FUNCTION_BLOCK L0_8070Service (* FAGOR 8070 CNC service FB *)
  (* Standard: 61499-2; Description: This FB is the entry point of the CNC service *)
  (* Version 0.0, 2014-09-01, EQUEROL, UJI *)
  (* Version 1.0, 2015-03-03, EQUEROL, UJI, Service rework *)
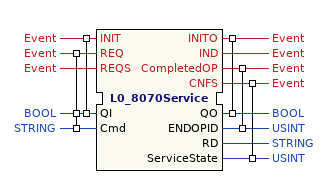
  EVENT_INPUT
    INIT WITH QI; (* Initialization Request *)
    REQ WITH QI, Cmd; (* Normal Execution Request *)
    REQS; (* Request Service state *)
  END_EVENT
  EVENT_OUTPUT
    INITO WITH QO; (* Initialization Confirm *)
    IND; (* Operation reception confirmation *)
    CompletedOP WITH ENDOPID; (* Completed operation event *)
    CNFS WITH ServiceState; (* Service State Confirmation *)
  END_EVENT
  VAR_INPUT
    QI : BOOL; (* Input event qualifier *)
    Cmd : STRING; (* String containing the actions to be executed *)
  END_VAR
  VAR_OUTPUT
    QO : BOOL; (* Output event qualifier *)
    ENDOPID : USINT; (* Operation end code *)
    RD : STRING; (* Service feedback data *)
    ServiceState : USINT; (* CNC Service state *)
  END_VAR
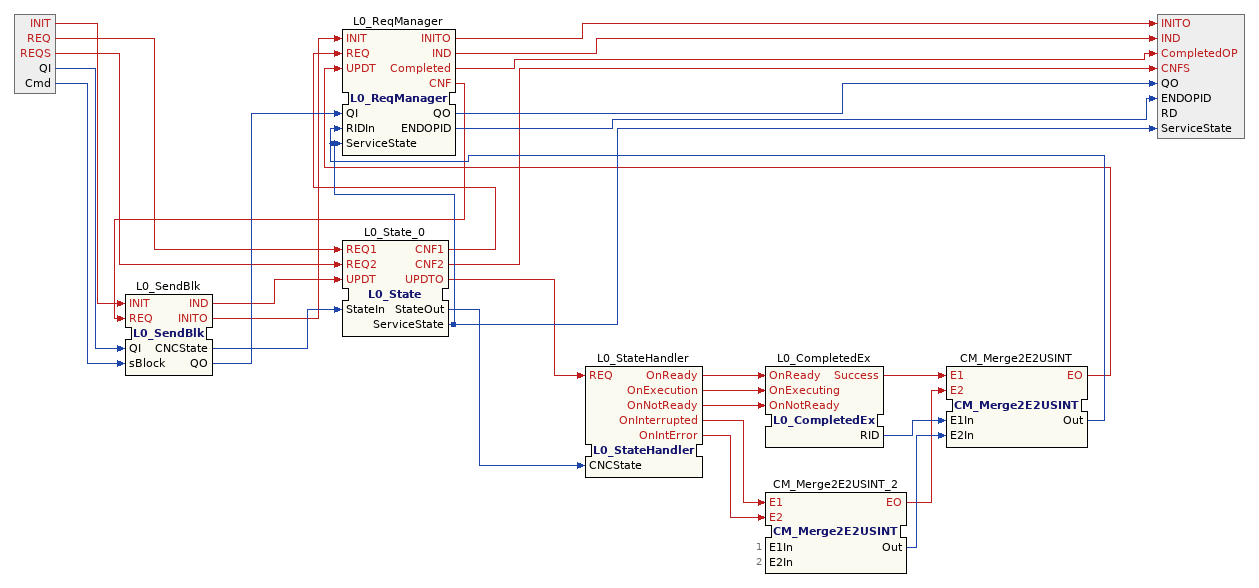
  FBS
    L0_SendBlk : L0_SendBlk;
    L0_StateHandler : L0_StateHandler;
    L0_CompletedEx : L0_CompletedEx;
    CM_Merge2E2USINT : CM_Merge2E2USINT;
    CM_Merge2E2USINT_2 : CM_Merge2E2USINT(E1In := 1, E2In := 2);
    L0_State_0 : L0_State;
    L0_ReqManager : L0_ReqManager;
  END_FBS
  EVENT_CONNECTIONS
    L0_StateHandler.OnReady TO L0_CompletedEx.OnReady;
    L0_StateHandler.OnExecution TO L0_CompletedEx.OnExecuting;
    L0_StateHandler.OnNotReady TO L0_CompletedEx.OnNotReady;
    L0_CompletedEx.Success TO CM_Merge2E2USINT.E1;
    CM_Merge2E2USINT_2.EO TO CM_Merge2E2USINT.E2;
    L0_StateHandler.OnInterrupted TO CM_Merge2E2USINT_2.E1;
    L0_StateHandler.OnIntError TO CM_Merge2E2USINT_2.E2;
    REQS TO L0_State_0.REQ2;
    L0_State_0.CNF2 TO CNFS;
    L0_State_0.UPDTO TO L0_StateHandler.REQ;
    L0_SendBlk.IND TO L0_State_0.UPDT;
    INIT TO L0_SendBlk.INIT;
    REQ TO L0_State_0.REQ1;
    L0_SendBlk.INITO TO L0_ReqManager.INIT;
    L0_State_0.CNF1 TO L0_ReqManager.REQ;
    CM_Merge2E2USINT.EO TO L0_ReqManager.UPDT;
    L0_ReqManager.INITO TO INITO;
    L0_ReqManager.CNF TO L0_SendBlk.REQ;
    L0_ReqManager.IND TO IND;
    L0_ReqManager.Completed TO CompletedOP;
  END_CONNECTIONS
  DATA_CONNECTIONS
    L0_CompletedEx.RID TO CM_Merge2E2USINT.E1In;
    CM_Merge2E2USINT_2.Out TO CM_Merge2E2USINT.E2In;
    L0_State_0.ServiceState TO ServiceState;
    L0_State_0.StateOut TO L0_StateHandler.CNCState;
    L0_SendBlk.CNCState TO L0_State_0.StateIn;
    QI TO L0_SendBlk.QI;
    L0_SendBlk.QO TO L0_ReqManager.QI;
    CM_Merge2E2USINT.Out TO L0_ReqManager.RIDIn;
    L0_ReqManager.QO TO QO;
    L0_ReqManager.ENDOPID TO ENDOPID;
    L0_State_0.ServiceState TO L0_ReqManager.ServiceState;
    Cmd TO L0_SendBlk.sBlock;
  END_CONNECTIONS
END_FUNCTION_BLOCK
